FUNCTION_BLOCK ILOCK_IO_AX (* Realizes a chainable momentary latch with interlock (AX/AX2 interface) *)
  (* Standard: 61499-1; Description: Copyright (c) 2026 Meisterschulen am Ostbahnhof *)
  (* Version 1.0, 2026-05-07, Gemini CLI, Meisterschulen am Ostbahnhof, initial version *)
  PACKAGE logiBUS::signalprocessing::interlock;
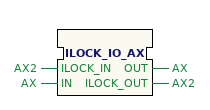
  SOCKETS
    ILOCK_IN : adapter::types::bidirectional::AX2; (* Interlock from above *)
    IN : adapter::types::unidirectional::AX; (* INPUT *)
  END_SOCKETS
  PLUGS
    OUT : adapter::types::unidirectional::AX; (* Output *)
    ILOCK_OUT : adapter::types::bidirectional::AX2; (* Interlock to below *)
  END_PLUGS
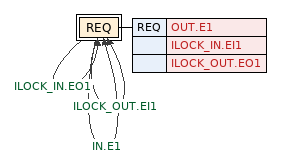
  EC_STATES
    REQ : REQ -> OUT.E1, -> ILOCK_IN.EI1, -> ILOCK_OUT.EO1;
  END_STATES
  EC_TRANSITIONS
    REQ TO REQ := IN.E1;
    REQ TO REQ := ILOCK_IN.EO1;
    REQ TO REQ := ILOCK_OUT.EI1;
  END_TRANSITIONS
  ALGORITHM REQ IN ST: (* Momentary latch: Q1 is active if SET is active AND no other element is set *)
OUT.D1 := IN.D1 AND NOT (ILOCK_IN.DO1 OR ILOCK_OUT.DI1);

(* Propagate status *)
ILOCK_IN.DI1 := OUT.D1;
ILOCK_OUT.DO1 := OUT.D1;
  END_ALGORITHM
END_FUNCTION_BLOCK
